// TIA Portal project "6_Assembler_Analog" (V19)

(* hardware
DEVICE "S7-1500/ET200MP station_1"  S7-1500 station
   slot 0: "Rail_0"  Rack  6ES7 590-1***0-0AA0
   slot 1: "PLC_1"  CPU 1513-1 PN  6ES7 513-1AL02-0AB0  V2.9
      slot 3: "CPU display_1"  6ES7591-1AA00-0AA0
      slot 32768: "PROFINET interface_1"  X1
         slot 32769: "Port_1"  X1 P1
         slot 32770: "Port_2"  X1 P2
      slot 34817: "Virtual CP interface port_1"  Virtual CP interface port  Virtual CP interface port
*)

// ===== PLC "PLC_1"  CPU 1513-1 PN =====

VAR_GLOBAL   // PLC tag table "Default tag table"
   "Tag_1" AT %M0.0 : Bool;
   "Tag_2" AT %M0.1 : Bool;
   "Tag_3" AT %M0.2 : Bool;
   "Tag_4" AT %M0.3 : Bool;
   "Tag_5" AT %M1.7 : Bool;
   "Tag_6" AT %M1.6 : Bool;
   "Tag_7" AT %M0.4 : Bool;
   "Tag_8" AT %M0.5 : Bool;
   "Tag_9" AT %M0.6 : Bool;
   "Tag_10" AT %M0.7 : Bool;
   "Tag_11" AT %M1.0 : Bool;
   "Tag_12" AT %M1.1 : Bool;
   "Tag_13" AT %M1.2 : Bool;
   "Tag_14" AT %M1.5 : Bool;
   "Tag_15" AT %M2.1 : Bool;
   "Tag_16" AT %M1.3 : Bool;
   "Tag_17" AT %M2.0 : Bool;
   "Tag_18" AT %M1.4 : Bool;
END_VAR

VAR_GLOBAL   // PLC tag table "Tag table from XML_1"
   "Start Button 1" AT %I0.0 : Bool;
   "Stop Button 1" AT %I0.1 : Bool;
   "Base at place" AT %I0.2 : Bool;
   "Lid at place" AT %I0.3 : Bool;
   "Part leaving" AT %I0.4 : Bool;
   "Item detected" AT %I0.5 : Bool;
   "Bases conveyor 1" AT %Q0.0 : Bool;
   "Bases conveyor 2" AT %Q0.1 : Bool;
   "Lids conveyor 1" AT %Q0.2 : Bool;
   "Lids conveyor 2" AT %Q0.3 : Bool;
   "Start Button 1 (Light)" AT %Q0.4 : Bool;
   "Stop Button 1 (Light)" AT %Q0.5 : Bool;
   "Stop blade 1" AT %Q0.6 : Bool;
   "Stop blade 2" AT %Q0.7 : Bool;
   "Grab" AT %Q1.0 : Bool;
   "X" AT %ID30 : Real;
   "Z" AT %ID34 : Real;
   "Digital Display 1" AT %QD30 : DInt;
   "Set X" AT %QD34 : Real;
   "Set Z" AT %QD38 : Real;
END_VAR

// folder: System blocks/Program resources

DATA_BLOCK "IEC_Counter_0_DB"   // DB1
{ S7_Optimized_Access := 'TRUE' }
AUTHOR : Simatic
FAMILY : IEC
NAME : CNTR
VERSION : 1.0
// stored: InstanceOfName IEC_COUNTER
"IEC_COUNTER"
BEGIN
END_DATA_BLOCK

DATA_BLOCK "IEC_Timer_0_DB"   // DB2
{ S7_Optimized_Access := 'TRUE' }
AUTHOR : Simatic
FAMILY : IEC
NAME : IEC_TMR
VERSION : 1.0
// stored: InstanceOfName IEC_TIMER
"IEC_TIMER"
BEGIN
END_DATA_BLOCK

DATA_BLOCK "IEC_Timer_0_DB_1"   // DB3
{ S7_Optimized_Access := 'TRUE' }
AUTHOR : Simatic
FAMILY : IEC
NAME : IEC_TMR
VERSION : 1.0
// stored: InstanceOfName IEC_TIMER
"IEC_TIMER"
BEGIN
END_DATA_BLOCK

// folder: (top level)

ORGANIZATION_BLOCK "Main"   // OB1, LAD, ProgramCycle
TITLE = "Main Program Sweep (Cycle)"
{ S7_Optimized_Access := 'TRUE' }
VERSION : 0.1
   VAR_INPUT
      Initial_Call : Bool;   // Initial call of this OB
      Remanence : Bool;   // =True, if remanent data are available
   END_VAR
   VAR_TEMP   // added for the SCL form of the ladder/FBD networks
      _w1 : Bool;
      _w2 : Bool;
      _w3 : Bool;
   END_VAR
BEGIN

REGION Network 1: Start LED and Stop LED ON/OFF
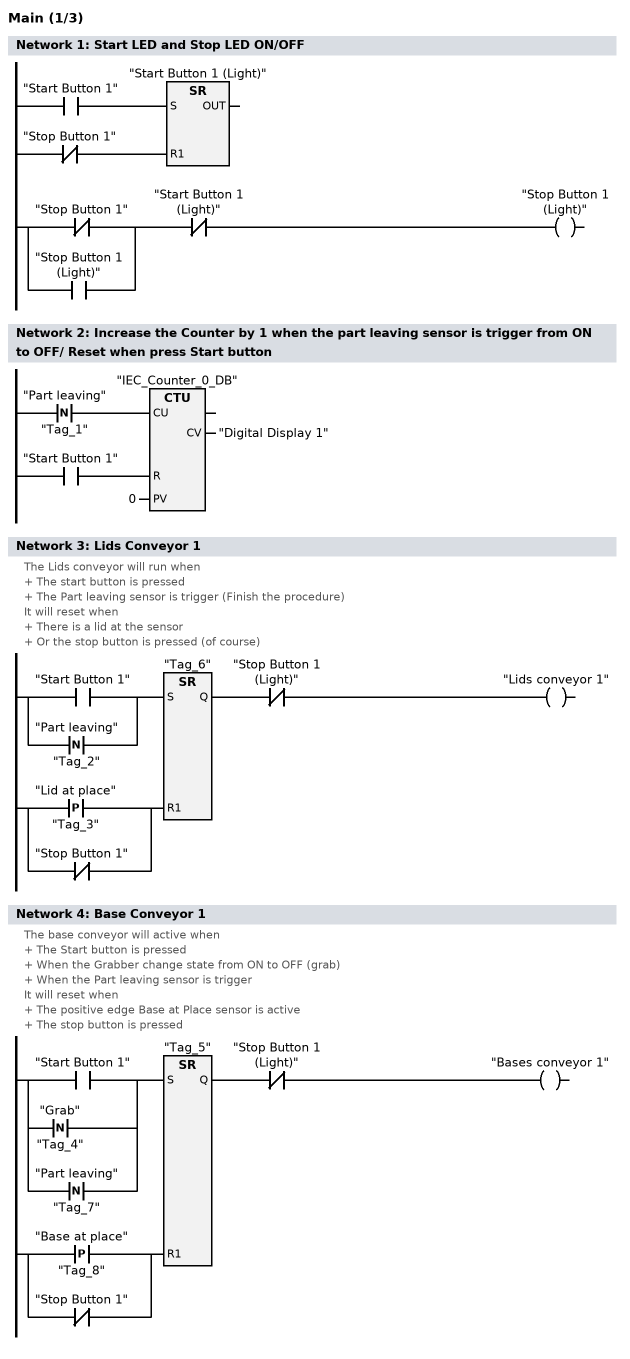
   RUNG wire#powerrail
      Contact( "Start Button 1" )
      S_SR(operand := "Start Button 1 (Light)", r1 := wire#w1)
   END_RUNG
   RUNG wire#powerrail
      I_Contact( "Stop Button 1" )
   END_RUNG wire#w1
   RUNG wire#powerrail
      I_Contact( "Stop Button 1" )
      wire#w2
      I_Contact( "Start Button 1 (Light)" )
      Coil( "Stop Button 1 (Light)" )
   END_RUNG
   RUNG wire#powerrail
      Contact( "Stop Button 1 (Light)" )
   END_RUNG wire#w2
   // the same network as SCL:
   IF "Start Button 1" THEN
       "Start Button 1 (Light)" := TRUE;   // SR flip-flop
   END_IF;
   IF NOT "Stop Button 1" THEN "Start Button 1 (Light)" := FALSE; END_IF;
   "Stop Button 1 (Light)" := (NOT "Stop Button 1" OR "Stop Button 1 (Light)") AND NOT "Start Button 1 (Light)";
END_REGION

REGION Network 2: Increase the Counter by 1 when the part leaving sensor is trigger from ON to OFF/ Reset when press Start button
   #_w1 := NOT "Part leaving" AND "Tag_1";   // falling edge of "Part leaving"
   "Tag_1" := "Part leaving";
   "IEC_Counter_0_DB".CTU(CU := #_w1, R := "Start Button 1", PV := 0, CV => "Digital Display 1");
END_REGION

REGION Network 3: Lids Conveyor 1
   // The Lids conveyor will run when
   // + The start button is pressed
   // + The Part leaving sensor is trigger (Finish the procedure)
   // It will reset when
   // + There is a lid at the sensor
   // + Or the stop button is pressed (of course)
   RUNG wire#powerrail
      Contact( "Start Button 1" )
      wire#w1
      S_SR(operand := "Tag_6", r1 := wire#w2)
      I_Contact( "Stop Button 1 (Light)" )
      Coil( "Lids conveyor 1" )
   END_RUNG
   RUNG wire#powerrail
      N_Contact(operand := "Part leaving", bit := "Tag_2")
   END_RUNG wire#w1
   RUNG wire#powerrail
      P_Contact(operand := "Lid at place", bit := "Tag_3")
   END_RUNG wire#w2
   RUNG wire#powerrail
      I_Contact( "Stop Button 1" )
   END_RUNG wire#w2
   // the same network as SCL:
   #_w1 := NOT "Part leaving" AND "Tag_2";   // falling edge of "Part leaving"
   "Tag_2" := "Part leaving";
   #_w2 := "Lid at place" AND NOT "Tag_3";   // rising edge of "Lid at place"
   "Tag_3" := "Lid at place";
   IF "Start Button 1" OR #_w1 THEN
       "Tag_6" := TRUE;   // SR flip-flop
   END_IF;
   IF #_w2 OR NOT "Stop Button 1" THEN "Tag_6" := FALSE; END_IF;
   "Lids conveyor 1" := "Tag_6" AND NOT "Stop Button 1 (Light)";
END_REGION

REGION Network 4: Base Conveyor 1
   // The base conveyor will active when
   // + The Start button is pressed
   // + When the Grabber change state from ON to OFF (grab)
   // + When the Part leaving sensor is trigger
   // It will reset when
   // + The positive edge Base at Place sensor is active
   // + The stop button is pressed
   RUNG wire#powerrail
      Contact( "Start Button 1" )
      wire#w1
      S_SR(operand := "Tag_5", r1 := wire#w2)
      I_Contact( "Stop Button 1 (Light)" )
      Coil( "Bases conveyor 1" )
   END_RUNG
   RUNG wire#powerrail
      N_Contact(operand := "Grab", bit := "Tag_4")
   END_RUNG wire#w1
   RUNG wire#powerrail
      N_Contact(operand := "Part leaving", bit := "Tag_7")
   END_RUNG wire#w1
   RUNG wire#powerrail
      P_Contact(operand := "Base at place", bit := "Tag_8")
   END_RUNG wire#w2
   RUNG wire#powerrail
      I_Contact( "Stop Button 1" )
   END_RUNG wire#w2
   // the same network as SCL:
   #_w1 := NOT "Grab" AND "Tag_4";   // falling edge of "Grab"
   "Tag_4" := "Grab";
   #_w2 := NOT "Part leaving" AND "Tag_7";   // falling edge of "Part leaving"
   "Tag_7" := "Part leaving";
   #_w3 := "Base at place" AND NOT "Tag_8";   // rising edge of "Base at place"
   "Tag_8" := "Base at place";
   IF "Start Button 1" OR #_w1 OR #_w2 THEN
       "Tag_5" := TRUE;   // SR flip-flop
   END_IF;
   IF #_w3 OR NOT "Stop Button 1" THEN "Tag_5" := FALSE; END_IF;
   "Bases conveyor 1" := "Tag_5" AND NOT "Stop Button 1 (Light)";
END_REGION

REGION Network 5: Base Conveyor 2
   // The base conveyor 2 will run when
   // + When the grabber change state from ON to OFF
   // and reset when
   // + The stop button is pressed
   // + The part leaving sensor is trigger negative edge create a line of product
   // + The start button is pressed
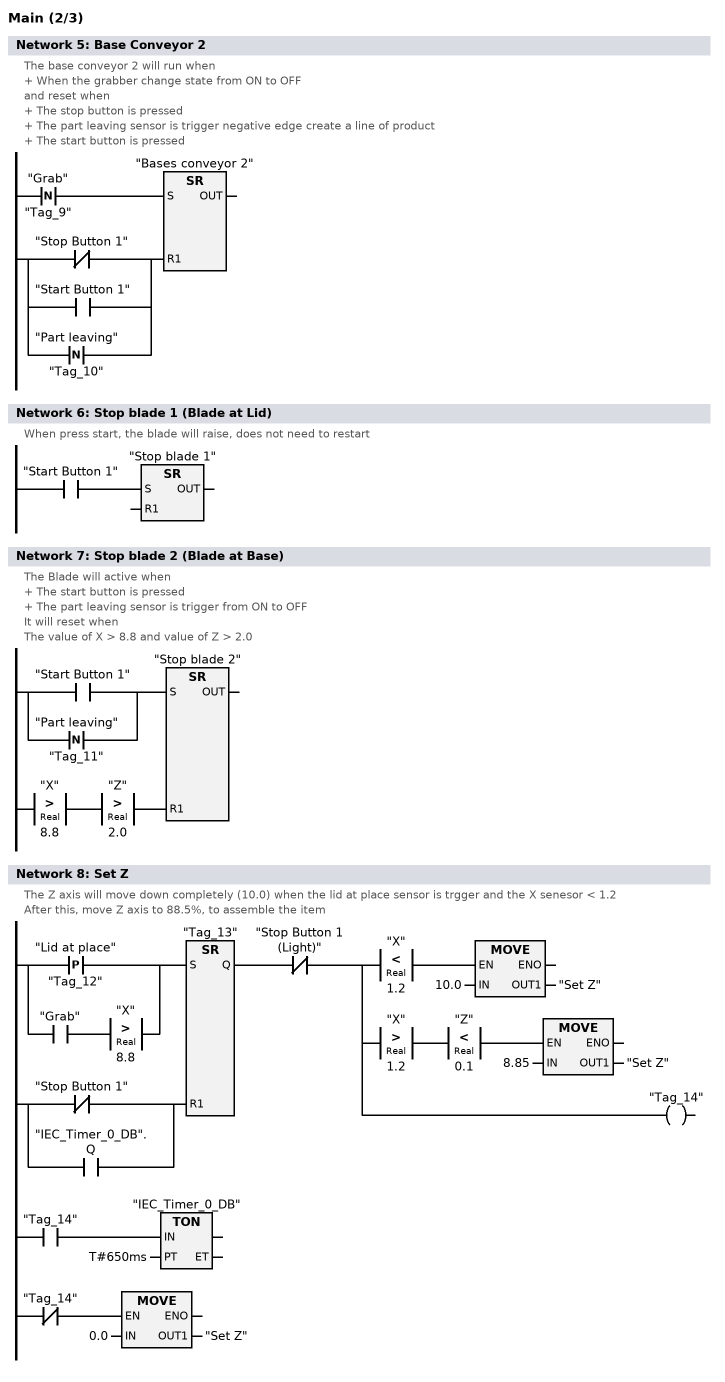
   RUNG wire#powerrail
      N_Contact(operand := "Grab", bit := "Tag_9")
      S_SR(operand := "Bases conveyor 2", r1 := wire#w1)
   END_RUNG
   RUNG wire#powerrail
      I_Contact( "Stop Button 1" )
   END_RUNG wire#w1
   RUNG wire#powerrail
      Contact( "Start Button 1" )
   END_RUNG wire#w1
   RUNG wire#powerrail
      N_Contact(operand := "Part leaving", bit := "Tag_10")
   END_RUNG wire#w1
   // the same network as SCL:
   #_w1 := NOT "Grab" AND "Tag_9";   // falling edge of "Grab"
   "Tag_9" := "Grab";
   #_w2 := NOT "Part leaving" AND "Tag_10";   // falling edge of "Part leaving"
   "Tag_10" := "Part leaving";
   IF #_w1 THEN
       "Bases conveyor 2" := TRUE;   // SR flip-flop
   END_IF;
   IF NOT "Stop Button 1" OR "Start Button 1" OR #_w2 THEN "Bases conveyor 2" := FALSE; END_IF;
END_REGION

REGION Network 6: Stop blade 1 (Blade at Lid)
   // When press start, the blade will raise, does not need to restart
   RUNG wire#powerrail
      Contact( "Start Button 1" )
      S_SR(operand := "Stop blade 1", r1 :=)
   END_RUNG
   // the same network as SCL:
   IF "Start Button 1" THEN
       "Stop blade 1" := TRUE;   // SR flip-flop
   END_IF;
END_REGION

REGION Network 7: Stop blade 2 (Blade at Base)
   // The Blade will active when
   // + The start button is pressed
   // + The part leaving sensor is trigger from ON to OFF
   // It will reset when
   // The value of X > 8.8 and value of Z > 2.0
   RUNG wire#powerrail
      Contact( "Start Button 1" )
      wire#w1
      S_SR(operand := "Stop blade 2", r1 := wire#w2)
   END_RUNG
   RUNG wire#powerrail
      N_Contact(operand := "Part leaving", bit := "Tag_11")
   END_RUNG wire#w1
   RUNG wire#powerrail
      { S7_Templates := "SrcType := Real" } GT_Contact(in1 := "X", in2 := 8.8)
      { S7_Templates := "SrcType := Real" } GT_Contact(in1 := "Z", in2 := 2.0)
   END_RUNG wire#w2
   // the same network as SCL:
   #_w1 := NOT "Part leaving" AND "Tag_11";   // falling edge of "Part leaving"
   "Tag_11" := "Part leaving";
   IF "Start Button 1" OR #_w1 THEN
       "Stop blade 2" := TRUE;   // SR flip-flop
   END_IF;
   IF ("X" > 8.8) AND ("Z" > 2.0) THEN "Stop blade 2" := FALSE; END_IF;
END_REGION

REGION Network 8: Set Z
   // The Z axis will move down completely (10.0) when the lid at place sensor is trgger and the X senesor < 1.2
   // After this, move Z axis to 88.5%, to assemble the item
   #_w1 := "Lid at place" AND NOT "Tag_12";   // rising edge of "Lid at place"
   "Tag_12" := "Lid at place";
   IF #_w1 OR ("Grab" AND ("X" > 8.8)) THEN
       "Tag_13" := TRUE;   // SR flip-flop
   END_IF;
   IF NOT "Stop Button 1" OR "IEC_Timer_0_DB".Q THEN "Tag_13" := FALSE; END_IF;
   #_w2 := "Tag_13" AND NOT "Stop Button 1 (Light)";
   IF #_w2 AND ("X" < 1.2) THEN "Set Z" := 10.0; END_IF;
   IF #_w2 AND ("X" > 1.2) AND ("Z" < 0.1) THEN "Set Z" := 8.85; END_IF;
   "Tag_14" := #_w2;
   "IEC_Timer_0_DB".TON(IN := "Tag_14", PT := T#650ms);
   IF NOT "Tag_14" THEN "Set Z" := 0.0; END_IF;
END_REGION

REGION Network 9: Grab
   // We need to work with network 8 at this moment.
   // The grab will turn on when the item detected sensor is ON, at the same time, the Z axis in network 8 will go down to pick the ojbect,
   // After that, the timer %DB2 will on and then move the Z-axis go up
   // The Grabber will leaves the item when %M1.5 in network 8 is activated and  Z-axis move down by 70%
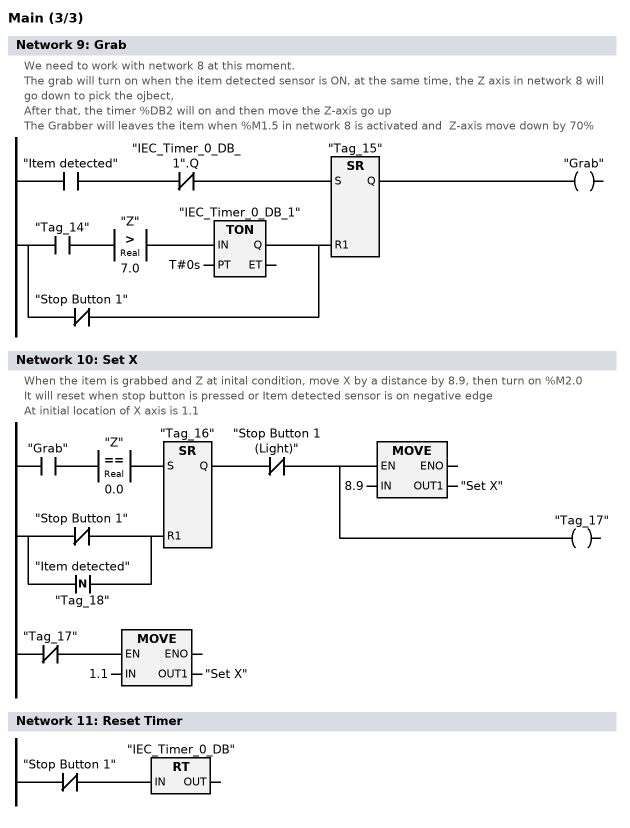
   #_w1 := "Item detected" AND NOT "IEC_Timer_0_DB_1".Q;
   "IEC_Timer_0_DB_1".TON(IN := "Tag_14" AND ("Z" > 7.0), PT := T#0s);
   IF #_w1 THEN
       "Tag_15" := TRUE;   // SR flip-flop
   END_IF;
   IF "IEC_Timer_0_DB_1".Q OR NOT "Stop Button 1" THEN "Tag_15" := FALSE; END_IF;
   "Grab" := "Tag_15";
END_REGION

REGION Network 10: Set X
   // When the item is grabbed and Z at inital condition, move X by a distance by 8.9, then turn on %M2.0
   // It will reset when stop button is pressed or Item detected sensor is on negative edge
   // At initial location of X axis is 1.1
   RUNG wire#powerrail
      Contact( "Grab" )
      { S7_Templates := "SrcType := Real" } EQ_Contact(in1 := "Z", in2 := 0.0)
      S_SR(operand := "Tag_16", r1 := wire#w1)
      I_Contact( "Stop Button 1 (Light)" )
      wire#w2
      Move(in := 8.9, out1 => "Set X")
   END_RUNG
   RUNG wire#powerrail
      I_Contact( "Stop Button 1" )
   END_RUNG wire#w1
   RUNG wire#powerrail
      N_Contact(operand := "Item detected", bit := "Tag_18")
   END_RUNG wire#w1
   RUNG wire#w2
      Coil( "Tag_17" )
   END_RUNG
   RUNG wire#powerrail
      I_Contact( "Tag_17" )
      Move(in := 1.1, out1 => "Set X")
   END_RUNG
   // the same network as SCL:
   #_w1 := NOT "Item detected" AND "Tag_18";   // falling edge of "Item detected"
   "Tag_18" := "Item detected";
   IF "Grab" AND ("Z" = 0.0) THEN
       "Tag_16" := TRUE;   // SR flip-flop
   END_IF;
   IF NOT "Stop Button 1" OR #_w1 THEN "Tag_16" := FALSE; END_IF;
   #_w2 := "Tag_16" AND NOT "Stop Button 1 (Light)";
   IF #_w2 THEN "Set X" := 8.9; END_IF;
   "Tag_17" := #_w2;
   IF NOT "Tag_17" THEN "Set X" := 1.1; END_IF;
END_REGION

REGION Network 11: Reset Timer
   RUNG wire#powerrail
      I_Contact( "Stop Button 1" )
      RT_Coil( "IEC_Timer_0_DB" )
   END_RUNG
   // the same network as SCL:
   IF NOT "Stop Button 1" THEN RESET_TIMER("IEC_Timer_0_DB"); END_IF;
END_REGION
END_ORGANIZATION_BLOCK